FUNCTION_BLOCK FB_ModulLogger IMPLEMENTS I_Logger
VAR_OUTPUT
	bAbort:						BOOL;
	bStop:						BOOL;
	bWarning:					BOOL;
	bInformation:				BOOL;
END_VAR

// Log events to the Module

METHOD M_Log
VAR_INPUT
	stEvent	: 		ST_Event;
END_VAR
IF stEvent.New THEN
	CASE stEvent.EventType OF
		E_Event.Error:
			IF stEvent.Command = 'Abort' THEN
				bAbort:= TRUE;		
			ELSIF stEvent.Command = 'Stop' THEN
				bStop:= TRUE;
			ELSIF stEvent.Command = 'StopCycle' THEN
				bStop:= TRUE;
			END_IF
	
		E_Event.Warning:
			bWarning:= TRUE;
			
		E_Event.Information:
			bInformation:= TRUE;
			
	END_CASE
END_IF
END_METHOD

END_FUNCTION_BLOCK

(* stored: Version 1.1.0.1
   POU FB_ModulLogger: Id {a5a249cb-e1f2-07f1-0e3a-a919b5fec1ea}, SpecialFunc None
   Method M_Log: Id {c003c572-188f-0727-0077-a74f5cfa4b92} *)
